// TIA Portal project "PLCSIM" (V16)

(* hardware
DEVICE "S71500/ET200MP station_1"  S7-1500 station
   slot 0: "导轨_0"  Rack  6ES7 590-1***0-0AA0
   slot 1: "PLC_1"  CPU 1511-1 PN  6ES7 511-1AK02-0AB0  V2.5
      slot 3: "CPU 显示_1"  6ES7591-1AA00-0AA0
      slot 32768: "PROFINET 接口_1"  X1
         slot 32769: "端口_1"  X1 P1
         slot 32770: "端口_2"  X1 P2
*)

// ===== PLC "PLC_1"  CPU 1511-1 PN =====

DATA_BLOCK "ModbusData"   // DB1
{ S7_Optimized_Access := 'FALSE' }
VERSION : 0.1
   VAR
      B0 : Bool;
      B1 : Bool;
      B2 : Bool;
      B3 : Bool;
      B4 : Bool;
      S0 : Int := 0;
      S1 : Int;
      S2 : Int;
      S3 : Int;
      S4 : Int;
      F0 : Real;
      F1 : Real;
      F2 : Real;
      F3 : Real;
      F4 : Real;
      Str0 : String[50];
      Str1 : String[50];
   END_VAR
BEGIN
END_DATA_BLOCK

DATA_BLOCK "ConnData"   // DB3
{ S7_Optimized_Access := 'TRUE' }
VERSION : 0.1
   VAR
      Conn : TCON_IP_v4;
   END_VAR
BEGIN
   Conn.ID := 16#1;
   Conn.LocalPort := 502;
   Conn.InterfaceId := 64;
END_DATA_BLOCK

ORGANIZATION_BLOCK "Main"   // OB1, LAD, ProgramCycle
TITLE = "Main Program Sweep (Cycle)"
{ S7_Optimized_Access := 'TRUE' }
VERSION : 0.1
   VAR_INPUT
      Initial_Call : Bool;   // Initial call of this OB
      Remanence : Bool;   // =True, if remanent data are available
   END_VAR
BEGIN

REGION Network 1
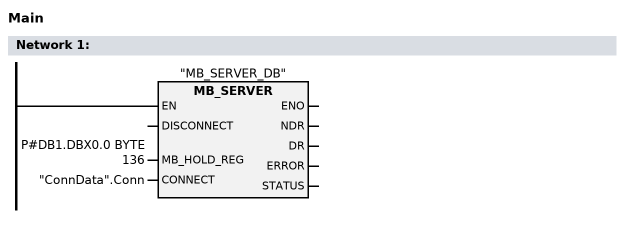
   "MB_SERVER_DB"(MB_HOLD_REG := P#DB1.DBX0.0 BYTE 136, CONNECT := "ConnData".Conn);   // MB_SERVER
END_REGION
END_ORGANIZATION_BLOCK